FUNCTION_BLOCK Test_F_TimeAsString_ms_ReturnsString_ms EXTENDS T_UnitTestBase
VAR
    TimeStruct : TIMESTRUCT := (wHour := 6, wMinute := 5, wSecond := 4, wMilliseconds := 135);
END_VAR

{attribute 'analysis' := '-33'} // inhibit unused variable warning
METHOD RunTest
IF Retest THEN
	SUPER^.Init();
END_IF

IF TestCompleted THEN
	RETURN;
END_IF

AssertEquals_STRING(Expected := '06:05:04.135',
                    Actual   := F_TimeAsString_ms(TimeStruct),
                    Message  := 'F_TimeAsString_ms(TimeStruct)');

TestCompleted := TRUE;
END_METHOD

END_FUNCTION_BLOCK

(* stored: Version 1.1.0.1, ProductVersion 3.1.4024.12
   POU Test_F_TimeAsString_ms_ReturnsString_ms: Id {cfe81a32-3eca-0666-0352-ea68d5a05067}, SpecialFunc None
   Method RunTest: Id {64e2b548-2cb6-0d36-03bb-73f3ee98bfe2} *)
